{attribute 'linkalways'} 
{attribute 'no_explicit_call' := 'This FB is a CLASS and must be accessed using methods or properties'}
{attribute 'enable_dynamic_creation'}
FUNCTION_BLOCK Node_F_VN_ImageMoments EXTENDS VisionNode
VAR
    ipImage : _ITcVnImage;
    stMoments : _TcVnMoments;
    bBinaryImage : _BOOL(FALSE);
    hrPrev : _HRESULT(S_OK);
	hresult : _HRESULT(S_OK);
END_VAR

METHOD PUBLIC  Clone : I_Node
VAR
	pNode : POINTER TO Node_F_VN_ImageMoments;
END_VAR
pNode := __NEW(Node_F_VN_ImageMoments);
Clone := pNode^;
END_METHOD

METHOD FB_init : BOOL
VAR_INPUT
	bInitRetains : BOOL; // if TRUE, the retain variables are initialized (warm start / cold start)
	bInCopyCode : BOOL;  // if TRUE, the instance afterwards gets moved into the copy code (online change)
END_VAR
AddInput('ipImage', ipImage);
AddParameter('bBinaryImage', bBinaryImage);
AddInput('hrPrev', hrPrev);
AddOutput('stMoments', stMoments);
AddOutput('hresult', hresult);
END_METHOD

METHOD PROTECTED OnExecute
hresult.Value := F_VN_ImageMoments(
	ipImage := ipImage.Value,
    stMoments := stMoments.Value,
    bBinaryImage := bBinaryImage.Value,
	hrPrev:= hrPrev.Value);
END_METHOD

METHOD PUBLIC PreExecutionCheck
VAR_INPUT
	Check : I_PreExecutionChecks;
END_VAR
Check.IsTrue(ipImage.IsValid, 'ipImage must contain an image');
Check.IsTrue(ipImage.HasChannelCount(1), 'ipImage must contain 1 channel');
Check.IsTrue((ipImage.IsPixelDepth(8) OR ipImage.IsPixelDepth(32)), 'ipImage must have 8 or 32 bit pixel depth');
END_METHOD

END_FUNCTION_BLOCK

(* stored: Version 1.1.0.1, ProductVersion 3.1.4024.13
   POU Node_F_VN_ImageMoments: Id {78908e80-3339-05c1-0be1-024fb003abb3}, SpecialFunc None
   Folder Constructor: Id {f998062d-21de-0ae1-22e6-001d58f69e83}
   Method Clone: Id {38949002-1e04-03fd-0481-3cbfceef5d3b}
   Method FB_init: Id {1e6914f9-bc84-00b5-0621-276cc6a30f2f}
   Method OnExecute: Id {4f0e92ad-1459-0b23-1b92-ba40b6fa575d}
   Method PreExecutionCheck: Id {ce031da2-fc70-04fd-0f7b-6297768f6b15} *)
